FUNCTION_BLOCK FB_HE_SATT_FilterTestDouble IMPLEMENTS I_HE_SATT_Filter
VAR
    iHolder : I_HE_SATT_FilterHolder;
    fLength : LREAL;
    eMaterial : E_HE_SATT_FilterMaterial;
    fPositionInHolder : LREAL;
    eStatus : E_HE_SATT_FilterStatus;
END_VAR


PROPERTY Holder : I_HE_SATT_FilterHolder
GET

Holder := THIS^.iHolder;
END_GET
SET

THIS^.iHolder := Holder;
END_SET
END_PROPERTY


PROPERTY Length : LREAL
GET

Length := THIS^.fLength;
END_GET
SET

THIS^.fLength := Length;
END_SET
END_PROPERTY


PROPERTY Material : E_HE_SATT_FilterMaterial
GET

Material := THIS^.eMaterial;
END_GET
SET

THIS^.eMaterial := Material;
END_SET
END_PROPERTY


PROPERTY PositionInHolder : LREAL
GET

PositionInHolder := THIS^.fPositionInHolder;
END_GET
SET

THIS^.fPositionInHolder := PositionInHolder;
END_SET
END_PROPERTY


PROPERTY Status : E_HE_SATT_FilterStatus
GET

Status := THIS^.eStatus;
END_GET
SET

THIS^.eStatus := Status;
END_SET
END_PROPERTY

END_FUNCTION_BLOCK

(* stored: Version 1.1.0.1
   POU FB_HE_SATT_FilterTestDouble: Id {78e15cd5-2ad9-4e36-8049-41459bd3f9ff}, SpecialFunc None
   Property Holder: Id {36a88056-bfc1-4156-bf8f-9ebd187d96c5}
   Get Get: Id {258f7eac-4a17-40dd-8fee-e62cc47c80bc}
   Set Set: Id {5f1a7c2e-9baa-4822-80c8-368d615fbb6d}
   Property Length: Id {80d6f460-3dda-488b-acc8-c395f1fef9cf}
   Get Get: Id {948ab73f-d9d5-4816-8ac9-602575a7954b}
   Set Set: Id {63de0404-317b-48ed-a31a-37cad81f0a04}
   Property Material: Id {6ea46809-3b90-489c-8c6d-36817f6cc304}
   Get Get: Id {37ebdd02-cbb1-4174-babb-568b506bdb5c}
   Set Set: Id {ded793c4-3c47-4e91-863a-a722b926a8bd}
   Property PositionInHolder: Id {0922f6a8-3ed7-48ad-b27e-2120730cda7b}
   Get Get: Id {16c6a587-533c-47a5-abda-f59c4d091858}
   Set Set: Id {11157f5d-a0bd-41fd-b431-109fedd92de2}
   Property Status: Id {ef2b89b8-ff34-418f-8bd7-7cae8ad13291}
   Get Get: Id {7a4a7987-733b-44b1-a6d9-76aa51d09552}
   Set Set: Id {08d464be-7328-4fff-9b52-ba3023011098} *)
